// TwinCAT 3 PLC project _02_FactoryPattern
// ProgramVersion: 3.1.4023.0
// libraries:
//   Tc2_Standard, * (Beckhoff Automation GmbH)
//   Tc2_System, * (Beckhoff Automation GmbH)
//   Tc2_Utilities, * (Beckhoff Automation GmbH)
//   Tc3_Module, * (Beckhoff Automation GmbH)
// project tree:
//   Factory Method Pattern/Objects/DUTs/ E_OBJECTS.TcDUT, I_Object.TcIO, ST_ObjectDef.TcDUT
//   Factory Method Pattern/Objects/ FB_ObjectFactory.TcPOU
//   Factory Method Pattern/Objects/POUs/ FB_Cylinder.TcPOU, FB_Door.TcPOU, FB_EmptyObject.TcPOU, FB_Motor.TcPOU, FB_Object.TcPOU
//   Factory Method Pattern/ P_FactoryPattern.TcPOU
//   / MAIN.TcPOU, PlcTask.TcTTO
// (motion and I/O tree: see PLC project 13_decorator)
// real-time tasks:
//   TASK PlcTask: cycle T#10ms, priority 20, ADS port 350
// variable links:

CONFIGURATION _02_FactoryPattern
    RESOURCE PLC ON TwinCAT3
        TASK PlcTask(INTERVAL := T#10ms, PRIORITY := 20);
        PROGRAM MAIN WITH PlcTask : MAIN;
    END_RESOURCE
END_CONFIGURATION

// ---- Factory Method Pattern/Objects/DUTs/E_OBJECTS.TcDUT
{attribute 'qualified_only'}
TYPE E_OBJECTS :
(
	UNDEFINED := 0,
	CYLINDER,
	DOOR,
	MOTOR
);
END_TYPE

// ---- Factory Method Pattern/Objects/DUTs/ST_ObjectDef.TcDUT
TYPE ST_ObjectDef :
STRUCT
	sObjectID			: STRING := 'Error';
	eObjectType			: E_Objects := E_Objects.UNDEFINED;
	bReleaseIfExists	: BOOL := FALSE; // release the pointer if the pointer is already set
END_STRUCT
END_TYPE

// ---- Factory Method Pattern/Objects/DUTs/I_Object.TcIO
// Abstract class definition
INTERFACE I_Object

METHOD Destruct : BOOL
VAR_INPUT
END_VAR
END_METHOD

METHOD M_GetObjectDescription : STRING
VAR_INPUT
END_VAR
END_METHOD

METHOD M_Reset : BOOL
VAR_INPUT
END_VAR
END_METHOD

METHOD M_Start : BOOL
VAR_INPUT
END_VAR
END_METHOD

PROPERTY P_Status : DWORD
GET
END_GET
END_PROPERTY

END_INTERFACE

// ---- MAIN.TcPOU
PROGRAM MAIN
VAR
END_VAR

(* 
	GOF 		Define an interface for creating an object, but let subclasses decide which class
				to instantiate. Factory Method lets a class defer instantiation to subclasses.
*)
P_FactoryPattern();

END_PROGRAM

// ---- Factory Method Pattern/P_FactoryPattern.TcPOU
PROGRAM P_FactoryPattern
VAR
// *************** OBJECT FACTORY
	arrstObjects			: ARRAY[1..NUMBEROFOBJECTS] OF ST_ObjectDef := 
								[
								(sObjectID:='Motor 01',eObjectType:=E_Objects.MOTOR),
								(sObjectID:='Cylinder 01',eObjectType:=E_Objects.CYLINDER),
								(sObjectID:='Door 01',eObjectType:=E_Objects.DOOR),
								(sObjectID:='Cylinder 02',eObjectType:=E_Objects.CYLINDER),
								(sObjectID:='Motor 02',eObjectType:=E_Objects.MOTOR),
								(sObjectID:='Spare 01',eObjectType:=E_Objects.UNDEFINED,bReleaseIfExists:=TRUE)								
								];
	// Object factory creating the above defined objects
	fbObjectFactory			: FB_ObjectFactory;
	arrfbObjects			: ARRAY[1..NUMBEROFOBJECTS] OF FB_Object; 
	bInit					: BOOL := TRUE;
	// Test data retrieval	
	arrsObjectDescription	: ARRAY[1..NUMBEROFOBJECTS] OF STRING;
	i						: INT;	
	// test destructor
	bDestruct				: BOOL;
	nDestruct				: INT;
	
// *************** ROUTER
	// router info (memory consumption)
	fbGetRouterStatusInfo 	: FB_GetRouterStatusInfo;
	stTCRouterStatusInfo	: ST_TCRouterStatusInfo;
	memAvailable			: DWORD;
END_VAR
VAR CONSTANT
	NUMBEROFOBJECTS			: INT := 7;
END_VAR

// *************** OBJECT FACTORY
IF bInit	THEN
	// define the pointers to the objects in the array
	aObjectFactoring();	
	bInit 			:= FALSE;
END_IF

// test retrieve data from created objects
FOR i := 1 TO NUMBEROFOBJECTS DO
	arrsObjectDescription[i] := arrfbObjects[i].M_GetObjectDescription();	
END_FOR

// destroy objects / free memory
IF bDestruct		THEN
	IF nDestruct > 0 AND nDestruct <= NUMBEROFOBJECTS THEN
		arrfbObjects[nDestruct].Destruct();
	END_IF
	bDestruct := FALSE;
END_IF

// *************** ROUTER INFO
// router status
fbGetRouterStatusInfo(
	sNetId:= , 
	bExecute:= NOT fbGetRouterStatusInfo.bBusy, 
	tTimeout:= , 
	bBusy=> , 
	bError=> , 
	nErrID=> , 
	info=> stTCRouterStatusInfo
	);
IF stTCRouterStatusInfo.maxMemAvail	> 0 THEN
	memAvailable := stTCRouterStatusInfo.maxMemAvail;
END_IF

ACTION aObjectFactoring:
// loop through definitions and create instances
FOR i := 1 TO NUMBEROFOBJECTS	DO
	fbObjectFactory(
		stObjectDef		:=arrstObjects[i], 
		fbObject		:=arrfbObjects[i]);
END_FOR
END_ACTION

END_PROGRAM

// ---- Factory Method Pattern/Objects/FB_ObjectFactory.TcPOU
FUNCTION_BLOCK FB_ObjectFactory
VAR_INPUT
	stObjectDef			: ST_ObjectDef;
END_VAR
VAR_IN_OUT
	fbObject 			: FB_Object;	// reference to the actual object
END_VAR
VAR
	pEmptyObject    	: POINTER TO FB_EmptyObject;
	pDoor       		: POINTER TO FB_Door;
	pCylinder   		: POINTER TO FB_Cylinder;
	pMotor       		: POINTER TO FB_Motor;			
END_VAR


// release pointer if existing
IF fbObject.ipObject <> 0 THEN
	IF stObjectDef.bReleaseIfExists	THEN
		// DONKEY First release before proceeding
		Destruct(fbObject); 
	ELSE
		// only proceed if there isn't already a pointer in ipObject
		RETURN;
	END_IF
END_IF

// return an instance reference to the requested object type 
CASE stObjectDef.eObjectType			OF
	
	E_OBJECTS.UNDEFINED:
		// create a pointer to the object to be instantiated				
		pEmptyObject  		:= __NEW(FB_EmptyObject(
								sObjectID		:=stObjectDef.sObjectID, 
								eObjectType		:=stObjectDef.eObjectType)
								);
		pEmptyObject^.pInstance := pEmptyObject; 	// store pointer for destructor						
		fbObject.ipObject	:= pEmptyObject^;		// reference pointer to the real FB
		
	E_OBJECTS.CYLINDER:
		pCylinder  			:= __NEW(FB_Cylinder(
								sObjectID		:=stObjectDef.sObjectID, 
								eObjectType		:=stObjectDef.eObjectType)
								);
		pCylinder^.pInstance := pCylinder; 							
		fbObject.ipObject	:= pCylinder^;
	
	E_OBJECTS.DOOR:
		pDoor	  			:= __NEW(FB_Door(
								sObjectID		:=stObjectDef.sObjectID, 
								eObjectType		:=stObjectDef.eObjectType)
								);
		pDoor^.pInstance	:= pDoor;
		fbObject.ipObject	:= pDoor^;
		
	E_OBJECTS.MOTOR:
		pMotor  			:= __NEW(FB_Motor(
								sObjectID		:=stObjectDef.sObjectID, 
								eObjectType		:=stObjectDef.eObjectType)
								);
		pMotor^.pInstance	:= pMotor;
		fbObject.ipObject	:= pMotor^;
		
	ELSE
		pEmptyObject  		:= __NEW(FB_EmptyObject(
								sObjectID		:='INVALID TYPE', 
								eObjectType		:=E_Objects.UNDEFINED)
								);
		pEmptyObject^.pInstance := pEmptyObject;						
		fbObject.ipObject	:= pEmptyObject^;
	
END_CASE

METHOD Destruct : BOOL
VAR_INPUT
	fbObject		: FB_Object;
END_VAR
fbObject.Destruct();
END_METHOD

END_FUNCTION_BLOCK

// ---- Factory Method Pattern/Objects/POUs/FB_Object.TcPOU
FUNCTION_BLOCK FB_Object IMPLEMENTS I_Object
VAR_INPUT
END_VAR
VAR_OUTPUT
END_VAR
VAR
	_ipObject 			: I_Object := 0;
END_VAR

METHOD Destruct : BOOL
// object destructor
IF (_ipObject <> 0) THEN
	_ipObject.Destruct();
	_ipObject := 16#0;
END_IF
END_METHOD

PROPERTY ipObject : I_Object
GET
ipObject := this^._ipObject;
END_GET
SET
IF (ipObject<>0) THEN
	THIS^._ipObject := ipObject;
ELSE
	THIS^._ipObject := 0;
END_IF
END_SET
END_PROPERTY

METHOD M_GetObjectDescription : STRING
M_GetObjectDescription := 'Error';
IF (_ipObject <> 0) THEN
	M_GetObjectDescription := _ipObject.M_GetObjectDescription();
END_IF
END_METHOD

{warning 'add method implementation'}
METHOD M_Reset : BOOL
END_METHOD

{warning 'add method implementation'}
METHOD M_Start : BOOL
END_METHOD

{warning 'add property implementation'}
PROPERTY P_Status : DWORD
GET
END_GET
END_PROPERTY

END_FUNCTION_BLOCK

// ---- Factory Method Pattern/Objects/POUs/FB_EmptyObject.TcPOU
{attribute 'enable_dynamic_creation'}
FUNCTION_BLOCK FB_EmptyObject IMPLEMENTS I_Object
VAR_INPUT
END_VAR
VAR_OUTPUT
END_VAR
VAR
	sObjectID			: STRING;
	eObjectType			: E_OBJECTS;
	// pointers for destructor
	_pInstance			: POINTER TO FB_EmptyObject;
	_pTemp				: POINTER TO FB_EmptyObject;
END_VAR

METHOD Destruct : BOOL
// destroy the instance 
IF _pInstance	<> 0 THEN
	// store in temp value otherwise the FB_exit called at __DELETE will create a stack overflow
	// when not set to 0 before __DELETE  
	_pTemp := _pInstance;
	_pInstance := 16#0; 
	__DELETE(_pTemp);
END_IF
END_METHOD

METHOD FB_exit : BOOL
VAR_INPUT
	bInCopyCode : BOOL; // if TRUE, the exit method is called for exiting an instance that is copied afterwards (online change).
END_VAR
Destruct();
END_METHOD

METHOD FB_init : BOOL
VAR_INPUT
	bInitRetains       : BOOL; // if TRUE, the retain variables are initialized (warm start / cold start)
	bInCopyCode        : BOOL;  // if TRUE, the instance afterwards gets moved into the copy code (online change)
	// Object identifier name
	sObjectID			: STRING;	
	// Object type as a string
	eObjectType			: E_OBJECTS;
END_VAR
THIS^.sObjectID		:= sObjectID;
THIS^.eObjectType	:= eObjectType;
END_METHOD

METHOD M_GetObjectDescription : string
VAR_INPUT
END_VAR
VAR
	sDescription			: STRING;
END_VAR
sDescription := concat(THIS^.sObjectID, ' Type: '); 
sDescription := concat(sDescription, TO_STRING(THIS^.eObjectType)); 
M_GetObjectDescription := sDescription;
END_METHOD

{warning 'add method implementation'}
METHOD M_Reset : BOOL
END_METHOD

{warning 'add method implementation'}
METHOD M_Start : BOOL
END_METHOD

{warning 'add property implementation'}
PROPERTY P_Status : DWORD
GET
END_GET
END_PROPERTY

PROPERTY pInstance : POINTER TO FB_EmptyObject
SET
// Store pointer for destructor
_pInstance := pInstance;
END_SET
END_PROPERTY

END_FUNCTION_BLOCK

// ---- Factory Method Pattern/Objects/POUs/FB_Door.TcPOU
{attribute 'enable_dynamic_creation'}
FUNCTION_BLOCK FB_Door IMPLEMENTS I_Object
VAR_INPUT
END_VAR
VAR_OUTPUT
END_VAR
VAR
	sObjectID			: STRING;
	eObjectType			: E_OBJECTS;
	// pointers for destructor
	_pInstance			: POINTER TO FB_Door;
	_pTemp				: POINTER TO FB_Door;
END_VAR

METHOD Destruct : BOOL
// destroy the instance 
IF _pInstance	<> 0 THEN
	// store in temp value otherwise the FB_exit called at __DELETE will create a stack overflow
	// when not set to 0 before __DELETE  
	_pTemp := _pInstance;
	_pInstance := 16#0; 
	__DELETE(_pTemp);
END_IF
END_METHOD

METHOD FB_init : BOOL
VAR_INPUT
	bInitRetains       : BOOL; // if TRUE, the retain variables are initialized (warm start / cold start)
	bInCopyCode        : BOOL;  // if TRUE, the instance afterwards gets moved into the copy code (online change)
	// Object identifier name
	sObjectID			: STRING;	
	// Object type as a string
	eObjectType			: E_OBJECTS;
END_VAR
THIS^.sObjectID		:= sObjectID;
THIS^.eObjectType	:= eObjectType;
END_METHOD

METHOD M_GetObjectDescription : string
VAR_INPUT
END_VAR
VAR
	sDescription			: STRING;
END_VAR
sDescription := concat(THIS^.sObjectID, ' Type: '); 
sDescription := concat(sDescription, TO_STRING(THIS^.eObjectType)); 
M_GetObjectDescription := sDescription;
END_METHOD

{warning 'add method implementation'}
METHOD M_Reset : BOOL
END_METHOD

{warning 'add method implementation'}
METHOD M_Start : BOOL
END_METHOD

{warning 'add property implementation'}
PROPERTY P_Status : DWORD
GET
END_GET
END_PROPERTY

PROPERTY pInstance : POINTER TO FB_EmptyObject
SET
// Store pointer for destructor
_pInstance := pInstance;
END_SET
END_PROPERTY

END_FUNCTION_BLOCK

// ---- Factory Method Pattern/Objects/POUs/FB_Cylinder.TcPOU
{attribute 'enable_dynamic_creation'}
FUNCTION_BLOCK FB_Cylinder IMPLEMENTS I_Object
VAR_INPUT
END_VAR
VAR_OUTPUT
END_VAR
VAR
	sObjectID			: STRING;
	eObjectType			: E_OBJECTS;
	// pointers for destructor
	_pInstance			: POINTER TO FB_Cylinder;
	_pTemp				: POINTER TO FB_Cylinder;
END_VAR

METHOD Destruct : BOOL
// destroy the instance 
IF _pInstance	<> 0 THEN
	// store in temp value otherwise the FB_exit called at __DELETE will create a stack overflow
	// when not set to 0 before __DELETE  
	_pTemp := _pInstance;
	_pInstance := 16#0; 
	__DELETE(_pTemp);
END_IF
END_METHOD

METHOD FB_init : BOOL
VAR_INPUT
	bInitRetains       : BOOL; // if TRUE, the retain variables are initialized (warm start / cold start)
	bInCopyCode        : BOOL;  // if TRUE, the instance afterwards gets moved into the copy code (online change)
	// Object identifier name
	sObjectID			: STRING;	
	// Object type as a string
	eObjectType			: E_OBJECTS;
END_VAR
THIS^.sObjectID		:= sObjectID;
THIS^.eObjectType	:= eObjectType;
END_METHOD

METHOD M_GetObjectDescription : string
VAR_INPUT
END_VAR
VAR
	sDescription			: STRING;
END_VAR
sDescription := concat(THIS^.sObjectID, ' Type: '); 
sDescription := concat(sDescription, TO_STRING(THIS^.eObjectType)); 
M_GetObjectDescription := sDescription;
END_METHOD

{warning 'add method implementation'}
METHOD M_Reset : BOOL
END_METHOD

{warning 'add method implementation'}
METHOD M_Start : BOOL
END_METHOD

{warning 'add property implementation'}
PROPERTY P_Status : DWORD
GET
END_GET
END_PROPERTY

PROPERTY pInstance : POINTER TO FB_EmptyObject
SET
// Store pointer for destructor
_pInstance := pInstance;
END_SET
END_PROPERTY

END_FUNCTION_BLOCK

// ---- Factory Method Pattern/Objects/POUs/FB_Motor.TcPOU
{attribute 'enable_dynamic_creation'}
FUNCTION_BLOCK FB_Motor IMPLEMENTS I_Object
VAR_INPUT
END_VAR
VAR_OUTPUT
END_VAR
VAR
	sObjectID			: STRING;
	eObjectType			: E_OBJECTS;
	// pointers for destructor
	_pInstance			: POINTER TO FB_Motor;
	_pTemp				: POINTER TO FB_Motor;
END_VAR

METHOD Destruct : BOOL
// destroy the instance 
IF _pInstance	<> 0 THEN
	// store in temp value otherwise the FB_exit called at __DELETE will create a stack overflow
	// when not set to 0 before __DELETE  
	_pTemp := _pInstance;
	_pInstance := 16#0; 
	__DELETE(_pTemp);
END_IF
END_METHOD

METHOD FB_init : BOOL
VAR_INPUT
	bInitRetains       : BOOL; // if TRUE, the retain variables are initialized (warm start / cold start)
	bInCopyCode        : BOOL;  // if TRUE, the instance afterwards gets moved into the copy code (online change)
	// Object identifier name
	sObjectID			: STRING;	
	// Object type as a string
	eObjectType			: E_OBJECTS;
END_VAR
THIS^.sObjectID		:= sObjectID;
THIS^.eObjectType	:= eObjectType;
END_METHOD

METHOD M_GetObjectDescription : string
VAR_INPUT
END_VAR
VAR
	sDescription			: STRING;
END_VAR
sDescription := concat(THIS^.sObjectID, ' Type: '); 
sDescription := concat(sDescription, TO_STRING(THIS^.eObjectType)); 
M_GetObjectDescription := sDescription;
END_METHOD

{warning 'add method implementation'}
METHOD M_Reset : BOOL
END_METHOD

{warning 'add method implementation'}
METHOD M_Start : BOOL
END_METHOD

{warning 'add property implementation'}
PROPERTY P_Status : DWORD
GET
END_GET
END_PROPERTY

PROPERTY pInstance : POINTER TO FB_EmptyObject
SET
// Store pointer for destructor
_pInstance := pInstance;
END_SET
END_PROPERTY

END_FUNCTION_BLOCK
